(* IEC 61131-3 sources: Std_PalletMover/Class/MQTTClient_Interface (part 5) *)

      pResult^.aData[0]$UDINT := DiagnosticData.ComDiagnosis.udDMEntries;

    //-------------------------------------------------------------
    //TX Rate
    //-------------------------------------------------------------
    MQTTCLIENTINTERFACE_DIAGNOSTIC_NEWINST_GET_TX_RATE:

      pResult^.aData[0]$UDINT := DiagnosticData.ComDiagnosis.udTxRate;

    //-------------------------------------------------------------
    //RX Rate
    //-------------------------------------------------------------
    MQTTCLIENTINTERFACE_DIAGNOSTIC_NEWINST_GET_RX_RATE:

      pResult^.aData[0]$UDINT := DiagnosticData.ComDiagnosis.udRxRate;

    //-------------------------------------------------------------
    //Total RX Bytes
    //-------------------------------------------------------------
    MQTTCLIENTINTERFACE_DIAGNOSTIC_NEWINST_GET_RX_BYTES:

      pResult^.aData[0]$UDINT := DiagnosticData.ComDiagnosis.udTotalBytesRx;

    //-------------------------------------------------------------
    //Total TX Bytes
    //-------------------------------------------------------------
    MQTTCLIENTINTERFACE_DIAGNOSTIC_NEWINST_GET_TX_BYTES:

      pResult^.aData[0]$UDINT := DiagnosticData.ComDiagnosis.udTotalBytesTx;

  end_case;

END_FUNCTION

FUNCTION MQTTClient_Interface::Diagnostic_Event
	VAR_INPUT
		Event 	: t_e_DiagnosticLogTypes;
		udValue 	: UDINT;
	END_VAR

  //==============================================================
  //Based on the event that occurred, change the diagnostic data
  //==============================================================
  case Event of
    //----------------------------------------------------------
    //Reset the Diagnostic Values
    //----------------------------------------------------------
    DL_Reset:

      //Reset the timestamp
      DiagnosticData.udLastCalcTimestamp := ops.tAbsolute;

      //Clear Values
      SigCLib.MemSet( dst :=  #DiagnosticData.ComDiagnosis,
                      c   :=  0x00,
                      len :=  sizeof(DiagnosticData.ComDiagnosis));

      SigCLib.MemSet( dst :=  #DiagnosticData.TransferRateCalc,
                      c   :=  0x00,
                      len :=  sizeof(DiagnosticData.TransferRateCalc));

    //----------------------------------------------------------
    //Increment Connection Count
    //----------------------------------------------------------
    DL_Connect:

      DiagnosticData.ComDiagnosis.udConnect += 1;

    //----------------------------------------------------------
    //Connection Failed
    //----------------------------------------------------------
    DL_ConnectFail:

      DiagnosticData.ComDiagnosis.udConnectFail += 1;

    //----------------------------------------------------------
    //Connection Retried
    //----------------------------------------------------------
    DL_ConnectRetry:

      DiagnosticData.ComDiagnosis.udConnectRetry += 1;

    //----------------------------------------------------------
    //Connection Watchdog Timed out
    //----------------------------------------------------------
    DL_WatchdogTimeout:

      DiagnosticData.ComDiagnosis.udWDTimeout += 1;

    //----------------------------------------------------------
    //NotUsed
    //----------------------------------------------------------
    DL_NotUsed:

    //----------------------------------------------------------
    //Last Error Code Returned from MQTTClient
    //----------------------------------------------------------
    DL_LastErrorCode:

      DiagnosticData.ComDiagnosis.udLastRet := udValue;

    //----------------------------------------------------------
    //Number of errors returned from MQTTClient
    //----------------------------------------------------------
    DL_Error:

      DiagnosticData.ComDiagnosis.udFailRet += 1;

    //----------------------------------------------------------
    //Number of subscribe requests
    //----------------------------------------------------------
    DL_SubRequest:

      DiagnosticData.ComDiagnosis.udSubReqs += 1;

    //----------------------------------------------------------
    //Number of failed subscribe requests
    //----------------------------------------------------------
    DL_SubFail:

      DiagnosticData.ComDiagnosis.udSubFail += 1;

    //----------------------------------------------------------
    //Number of Publish Requests
    //----------------------------------------------------------
    DL_PubRequest:

      DiagnosticData.ComDiagnosis.udPubReq += 1;

    //----------------------------------------------------------
    //Number of failed Publishes
    //----------------------------------------------------------
    DL_PubFail:

      DiagnosticData.ComDiagnosis.udPubFail += 1;

    //----------------------------------------------------------
    //Number of Unsubscribe requests
    //----------------------------------------------------------
    DL_UnsubRequest:

      DiagnosticData.ComDiagnosis.udUnsubReq += 1;

    //----------------------------------------------------------
    //Unsubscribe Failed
    //----------------------------------------------------------
    DL_UnsubFail:

      DiagnosticData.ComDiagnosis.udUnsubFail += 1;

    //----------------------------------------------------------
    //Set PubSubEntries
    //----------------------------------------------------------
    DL_PubSubEntries:

      DiagnosticData.ComDiagnosis.udPubSubEntries := udValue;

    //----------------------------------------------------------
    //Add Log
    //----------------------------------------------------------
    DL_Log:

      DiagnosticData.ComDiagnosis.udLogs += 1;

    //----------------------------------------------------------
    //Ping Request Sent
    //----------------------------------------------------------
    DL_PingReq:

      DiagnosticData.ComDiagnosis.udPingReq += 1;

    //----------------------------------------------------------
    //Ping Response Received
    //----------------------------------------------------------
    DL_PingResp:

      DiagnosticData.ComDiagnosis.udPingResp += 1;

    //----------------------------------------------------------
    //QOS 0 Publish made
    //----------------------------------------------------------
    DL_Pub0:

      DiagnosticData.ComDiagnosis.udPubQOS0 += 1;

    //----------------------------------------------------------
    //QOS1 Publish Made
    //----------------------------------------------------------
    DL_Pub1:

      DiagnosticData.ComDiagnosis.udPubQOS1 += 1;

    //----------------------------------------------------------
    //QOS2 Publish Made
    //----------------------------------------------------------
    DL_Pub2:

      DiagnosticData.ComDiagnosis.udPubQOS2 += 1;

    //----------------------------------------------------------
    //QOS0 Subscribe Made
    //----------------------------------------------------------
    DL_Sub0:

      DiagnosticData.ComDiagnosis.udSubQOS0 += 1;

    //----------------------------------------------------------
    //QOS1 Subscribe Made
    //----------------------------------------------------------
    DL_Sub1:

      DiagnosticData.ComDiagnosis.udSubQOS1 += 1;

    //----------------------------------------------------------
    //QOS2 Subscribe Made
    //----------------------------------------------------------
    DL_Sub2:

      DiagnosticData.ComDiagnosis.udSubQOS2 += 1;

    //----------------------------------------------------------
    //Set DataMap Entries
    //----------------------------------------------------------
    DL_DataMapEntries:

      DiagnosticData.ComDiagnosis.udDMEntries := udValue;

    //----------------------------------------------------------
    //Set TX Rate
    //----------------------------------------------------------
    DL_TXRate:

      DiagnosticData.ComDiagnosis.udTxRate := udValue;

    //----------------------------------------------------------
    //Set RX Rate
    //----------------------------------------------------------
    DL_RXRate:

      DiagnosticData.ComDiagnosis.udRxRate := udValue;

    //----------------------------------------------------------
    //Set RX Bytes
    //----------------------------------------------------------
    DL_RXBytes:

      DiagnosticData.ComDiagnosis.udTotalBytesRx += udValue;

    //----------------------------------------------------------
    //Set TX Bytes
    //----------------------------------------------------------
    DL_TXBytes:

      DiagnosticData.ComDiagnosis.udTotalBytesTx += udValue;

  end_case;

END_FUNCTION

FUNCTION MQTTClient_Interface::ConfigObject_Process
	VAR_OUTPUT
		eRet 	: t_e_TaskRet;
	END_VAR
  VAR
  	ClientIDConfig          : MQTTClient_Interface_ConfigBase::t_s_ClientID;
    ConnectionDetailsConfig : MQTTClient_Interface_ConfigBase::t_s_ConnectionParameters;
    MIMConfig               : MQTTClient_Interface_ConfigBase::t_s_MaxInflightMessages;
    AuthenticationConfig    : MQTTClient_Interface_ConfigBase::t_s_Authentication;
    WillConfig              : MQTTClient_Interface_ConfigBase::t_s_Will;
    ReconnectionConfig      : MQTTClient_Interface_ConfigBase::t_s_ReconnectionParameters;
    TLSConfig               : MQTTClient_Interface_ConfigBase::t_s_TLS;
    tmpPara1                : DINT;
  END_VAR

  //Assume Busy
  eRet := TR_Busy;

  //======================================
  //Proccess the Config Object
  //======================================
  case Config.ConfigObject.State of
    //----------------------------
    //Client ID
    //----------------------------
    CO_ClientID:

      //Call the Config Method
      ClientIDConfig := Config.ConfigObject.pThis$^MQTTClient_Interface_ConfigBase^.ClientID();

      //Check if the config has been made, set the values
      if ClientIDConfig.ClientID <> ACCESS_DENIED then

        //If the input is OK, set the parameters
        if ClientIDConfig.ClientID                                                             &
           SigCLib.StrLen16(str0:=ClientIDConfig.ClientID) < MQTT_PROT_MAX_CLIENTID_NAME_LEN   then

          SigCLib.MemSet( dst   :=  #MQTTClientConfigData.Config.aClientID[0],
                          c     :=  0x00,
                          len   :=  sizeof(MQTTClientConfigData.Config.aClientID));
          SigCLib.StrCpy16(dst0 :=  #MQTTClientConfigData.Config.aClientID[0],
                           src0 :=  ClientIDConfig.ClientID);

          MQTTClientConfigData.Config.bClientIDSet := TRUE;

        //Input Not OK, Log
        else

          Logging_InterfLog(usLevel   :=  MQTTCLIENTINTERFACE_LOGGING_LEVEL_ERR,
                            dMsgGroup :=  MQCLIINF_LOG_ERROR_CONFIG_OBJ_CLIENTID_STRING_LEN_GRP,
                            dMsgNbr   :=  MQCLIINF_LOG_ERROR_CONFIG_OBJ_CLIENTID_STRING_LEN_MSG,
                            pMsg      :=  MQCLIINF_LOG_ERROR_CONFIG_OBJ_CLIENTID_STRING_LEN_TEXT,
                            pPara1    :=  NIL,
                            pPara2    :=  NIL,
                            pPara3    :=  NIL,
                            pPara4    :=  NIL);

        end_if;

      end_if;

      Config.ConfigObject.State := CO_ConnectionDetails;

    //----------------------------
    //Connection Details
    //----------------------------
    CO_ConnectionDetails:

      //Call the Config Method
      ConnectionDetailsConfig := Config.ConfigObject.pThis$^MQTTClient_Interface_ConfigBase^.ConnectionParameters();

      //Check if the config has been made
      if ConnectionDetailsConfig.hostname <> ACCESS_DENIED then

        //If the input is OK, set the parameters
        if ConnectionDetailsConfig.hostname                                                        &
           SigCLib.StrLen16(str0:=ConnectionDetailsConfig.hostname) < MQTTCLIENT_HOSTNAME_MAX_LEN  then

          SigCLib.MemSet( dst   :=  #MQTTClientConfigData.Config.Connect.aHostname[0],
                          c     :=  0x00,
                          len   :=  sizeof(MQTTClientConfigData.Config.Connect.aHostname));
          SigCLib.StrCpy16( dst0  :=  #MQTTClientConfigData.Config.Connect.aHostname[0],
                            src0  :=  ConnectionDetailsConfig.hostname);

          MQTTClientConfigData.Config.Connect.ValuesSet.Hostname := TRUE;

        //Input Not OK, Log
        else

          Logging_InterfLog(usLevel   :=  MQTTCLIENTINTERFACE_LOGGING_LEVEL_ERR,
                            dMsgGroup :=  MQCLIINF_LOG_ERROR_CONFIG_OBJ_HOSTNAME_STR_LEN_GRP,
                            dMsgNbr   :=  MQCLIINF_LOG_ERROR_CONFIG_OBJ_HOSTNAME_STR_LEN_MSG,
                            pMsg      :=  MQCLIINF_LOG_ERROR_CONFIG_OBJ_HOSTNAME_STR_LEN_TEXT,
                            pPara1    :=  NIL,
                            pPara2    :=  NIL,
                            pPara3    :=  NIL,
                            pPara4    :=  NIL);

        end_if;

        //If the input is OK, set the parameters
        if ConnectionDetailsConfig.port > 0       &
           ConnectionDetailsConfig.port <= 65536  then

          MQTTClientConfigData.Config.Connect.iPort := ConnectionDetailsConfig.port;
          MQTTClientConfigData.Config.Connect.ValuesSet.Port := TRUE;

        //Input Not OK, Log
        else

          tmpPara1 := to_dint(ConnectionDetailsConfig.port);

          Logging_InterfLog(usLevel   :=  MQTTCLIENTINTERFACE_LOGGING_LEVEL_ERR,
                            dMsgGroup :=  MQCLIINF_LOG_ERROR_CONFIG_OBJ_PORT_INVALID_GRP,
                            dMsgNbr   :=  MQCLIINF_LOG_ERROR_CONFIG_OBJ_PORT_INVALID_MSG,
                            pMsg      :=  MQCLIINF_LOG_ERROR_CONFIG_OBJ_PORT_INVALID_TEXT,
                            pPara1    :=  #tmpPara1,
                            pPara2    :=  NIL,
                            pPara3    :=  NIL,
                            pPara4    :=  NIL);

        end_if;

        //If the input is OK, set the parameters
        if ConnectionDetailsConfig.keepalive > 0       &
           ConnectionDetailsConfig.keepalive <= 65536  then

          MQTTClientConfigData.Config.Connect.iKeepalive := ConnectionDetailsConfig.keepalive;
          MQTTClientConfigData.Config.Connect.ValuesSet.Keepalive := TRUE;

        //Input Not OK, Log
        else

          tmpPara1 := to_dint(ConnectionDetailsConfig.keepalive);

          Logging_InterfLog(usLevel   :=  MQTTCLIENTINTERFACE_LOGGING_LEVEL_ERR,
                            dMsgGroup :=  MQCLIINF_LOG_ERROR_CONFIG_OBJ_KEEPALIVE_INVALID_GRP,
                            dMsgNbr   :=  MQCLIINF_LOG_ERROR_CONFIG_OBJ_KEEPALIVE_INVALID_MSG,
                            pMsg      :=  MQCLIINF_LOG_ERROR_CONFIG_OBJ_KEEPALIVE_INVALID_TEXT,
                            pPara1    :=  #tmpPara1,
                            pPara2    :=  NIL,
                            pPara3    :=  NIL,
                            pPara4    :=  NIL);

        end_if;

      end_if;

      Config.ConfigObject.State := CO_MaxInflightMessages;

    //----------------------------
    //Max Inflight Messages
    //----------------------------
    CO_MaxInflightMessages:

      //Call the Config Method
      MIMConfig := Config.ConfigObject.pThis$^MQTTClient_Interface_ConfigBase^.MaxInflightMessages();

      //Check if the config has been made
      if MIMConfig.max_inflight_messages <> -1 then

        //If the input is OK, set the parameters
        if MIMConfig.max_inflight_messages >= MQTTCLIENT_MIN_INFLIGHT_MSGS then

          MQTTClientConfigData.Config.Connect.iMaxInflightMessages  := MIMConfig.max_inflight_messages;
          MQTTClientConfigData.Config.Connect.ValuesSet.MaxInflight := TRUE;

        //Input Not OK, Log
        else

          tmpPara1 := MQTTCLIENT_MIN_INFLIGHT_MSGS;

          Logging_InterfLog(usLevel   :=  MQTTCLIENTINTERFACE_LOGGING_LEVEL_ERR,
                            dMsgGroup :=  MQCLIINF_LOG_ERROR_CONFIG_OBJ_MAX_INF_MSGS_LOW_GRP,
                            dMsgNbr   :=  MQCLIINF_LOG_ERROR_CONFIG_OBJ_MAX_INF_MSGS_LOW_MSG,
                            pMsg      :=  MQCLIINF_LOG_ERROR_CONFIG_OBJ_MAX_INF_MSGS_LOW_TEXT,
                            pPara1    :=  #tmpPara1,
                            pPara2    :=  NIL,
                            pPara3    :=  NIL,
                            pPara4    :=  NIL);

        end_if;

      end_if;

      Config.ConfigObject.State := CO_Authentication;

    //----------------------------
    //Authentication
    //----------------------------
    CO_Authentication:

      //Call the Config Method
      AuthenticationConfig := Config.ConfigObject.pThis$^MQTTClient_Interface_ConfigBase^.AuthenticationParameters();

      //Check if the config has been made
      if AuthenticationConfig.username <> ACCESS_DENIED then

        //If the input is OK, set the parameters
        if AuthenticationConfig.username                                                                         &
           SigCLib.StrLen16(str0:=AuthenticationConfig.username) < MQTTCLIENTINTERFACE_CONNECT_USERNAME_MAX_LEN  then

          SigCLib.MemSet( dst   :=  #MQTTClientConfigData.Config.Connect.aUsername[0],
                          c     :=  0x00,
                          len   :=  sizeof(MQTTClientConfigData.Config.Connect.aUsername));
          SigCLib.StrCpy16( dst0  :=  #MQTTClientConfigData.Config.Connect.aUsername[0],
                            src0  :=  AuthenticationConfig.username);

          MQTTClientConfigData.Config.Connect.ValuesSet.Username := TRUE;

        //Input Not OK, Log
        else

          tmpPara1 := MQTTCLIENTINTERFACE_CONNECT_USERNAME_MAX_LEN;

          Logging_InterfLog(usLevel   :=  MQTTCLIENTINTERFACE_LOGGING_LEVEL_ERR,
                            dMsgGroup :=  MQCLIINF_LOG_ERROR_CONFIG_OBJ_AUTH_USN_STR_LEN_GRP,
                            dMsgNbr   :=  MQCLIINF_LOG_ERROR_CONFIG_OBJ_AUTH_USN_STR_LEN_MSG,
                            pMsg      :=  MQCLIINF_LOG_ERROR_CONFIG_OBJ_AUTH_USN_STR_LEN_TEXT,
                            pPara1    :=  #tmpPara1,
                            pPara2    :=  NIL,
                            pPara3    :=  NIL,
                            pPara4    :=  NIL);

          MQTTClientConfigData.Config.Connect.ValuesSet.Username := FALSE;

        end_if;

        //If the input is OK, set the parameters
        if AuthenticationConfig.password                                                                         &
           SigCLib.StrLen16(str0:=AuthenticationConfig.password) < MQTTCLIENTINTERFACE_CONNECT_PASSWORD_MAX_LEN  then

          SigCLib.MemSet( dst   :=  #MQTTClientConfigData.Config.Connect.aPassword[0],
                          c     :=  0x00,
                          len   :=  sizeof(MQTTClientConfigData.Config.Connect.aPassword));
          SigCLib.StrCpy16( dst0  :=  #MQTTClientConfigData.Config.Connect.aPassword[0],
                            src0  :=  AuthenticationConfig.password);

          MQTTClientConfigData.Config.Connect.ValuesSet.Password := TRUE;

        //Input Not OK, Log
        else

          tmpPara1 := MQTTCLIENTINTERFACE_CONNECT_PASSWORD_MAX_LEN;

          Logging_InterfLog(usLevel   :=  MQTTCLIENTINTERFACE_LOGGING_LEVEL_ERR,
                            dMsgGroup :=  MQCLIINF_LOG_ERROR_CONFIG_OBJ_AUTH_PASS_STR_LEN_GRP,
                            dMsgNbr   :=  MQCLIINF_LOG_ERROR_CONFIG_OBJ_AUTH_PASS_STR_LEN_MSG,
                            pMsg      :=  MQCLIINF_LOG_ERROR_CONFIG_OBJ_AUTH_PASS_STR_LEN_TEXT,
                            pPara1    :=  #tmpPara1,
                            pPara2    :=  NIL,
                            pPara3    :=  NIL,
                            pPara4    :=  NIL);

          MQTTClientConfigData.Config.Connect.ValuesSet.Password := FALSE;

        end_if;

      end_if;

      Config.ConfigObject.State := CO_Will;

    //----------------------------
    //Will Config
    //----------------------------
    CO_Will:

      //Call the Config Method
      WillConfig := Config.ConfigObject.pThis$^MQTTClient_Interface_ConfigBase^.Will();

      //Check if the config has been made
      if WillConfig.topic <> ACCESS_DENIED then

        //If the input is OK, set the parameters
        if WillConfig.topic                                                                   &
           SigCLib.StrLen16(str0:=WillConfig.topic) < MQTTCLIENTINTERFACE_WILL_TOPIC_MAX_LEN  then

          SigCLib.MemSet( dst   :=  #MQTTClientConfigData.Config.Will.aTopic[0],
                          c     :=  0x00,
                          len   :=  sizeof(MQTTClientConfigData.Config.Will.aTopic));
          SigCLib.StrCpy16( dst0  :=  #MQTTClientConfigData.Config.Will.aTopic[0],
                            src0  :=  WillConfig.topic);

          MQTTClientConfigData.Config.Will.ValuesSet.Topic := TRUE;

        //Input Not OK, Log
        else

          tmpPara1 := MQTTCLIENTINTERFACE_WILL_TOPIC_MAX_LEN;

          Logging_InterfLog(usLevel   :=  MQTTCLIENTINTERFACE_LOGGING_LEVEL_ERR,
                            dMsgGroup :=  MQCLIINF_LOG_ERROR_CONFIG_OBJ_WILL_TOPIC_STR_LEN_GRP,
                            dMsgNbr   :=  MQCLIINF_LOG_ERROR_CONFIG_OBJ_WILL_TOPIC_STR_LEN_MSG,
                            pMsg      :=  MQCLIINF_LOG_ERROR_CONFIG_OBJ_WILL_TOPIC_STR_LEN_TEXT,
                            pPara1    :=  #tmpPara1,
                            pPara2    :=  NIL,
                            pPara3    :=  NIL,
                            pPara4    :=  NIL);

        end_if;

        //If the input is OK, set the parameters
        if WillConfig.payloadtext                                                                  &
           SigCLib.StrLen(str:=WillConfig.payloadtext) < MQTTCLIENTINTERFACE_WILL_PAYLOAD_MAX_LEN  then

          SigCLib.MemSet( dst   :=  #MQTTClientConfigData.Config.Will.aPayload[0],
                          c     :=  0x00,
                          len   :=  sizeof(MQTTClientConfigData.Config.Will.aPayload));
          SigCLib.StrCpy( dst0  :=  #MQTTClientConfigData.Config.Will.aPayload[0],
                          src0  :=  WillConfig.payloadtext);

          MQTTClientConfigData.Config.Will.ValuesSet.Payload := TRUE;

        //Input Not OK, Log
        else

          tmpPara1 := MQTTCLIENTINTERFACE_WILL_PAYLOAD_MAX_LEN;

          Logging_InterfLog(usLevel   :=  MQTTCLIENTINTERFACE_LOGGING_LEVEL_ERR,
                            dMsgGroup :=  MQCLIINF_LOG_ERROR_CONFIG_OBJ_WILL_PAYLOAD_STR_LEN_GRP,
                            dMsgNbr   :=  MQCLIINF_LOG_ERROR_CONFIG_OBJ_WILL_PAYLOAD_STR_LEN_MSG,
                            pMsg      :=  MQCLIINF_LOG_ERROR_CONFIG_OBJ_WILL_PAYLOAD_STR_LEN_TEXT,
                            pPara1    :=  #tmpPara1,
                            pPara2    :=  NIL,
                            pPara3    :=  NIL,
                            pPara4    :=  NIL);

        end_if;

        //If the input is OK, set the parameters
        if WillConfig.qos >= MQTT_PROT_QOS_MIN  &
           WillConfig.qos <= MQTT_PROT_QOS_MAX  then

          MQTTClientConfigData.Config.Will.iQoS := WillConfig.qos;
          MQTTClientConfigData.Config.Will.ValuesSet.QoS := TRUE;

        //Input Not OK, Log
        else

          tmpPara1 := to_dint(WillConfig.qos);

          Logging_InterfLog(usLevel   :=  MQTTCLIENTINTERFACE_LOGGING_LEVEL_ERR,
                            dMsgGroup :=  MQCLIINF_LOG_ERROR_CONFIG_OBJ_WILL_QOS_INVALID_GRP,
                            dMsgNbr   :=  MQCLIINF_LOG_ERROR_CONFIG_OBJ_WILL_QOS_INVALID_MSG,
                            pMsg      :=  MQCLIINF_LOG_ERROR_CONFIG_OBJ_WILL_QOS_INVALID_TEXT,
                            pPara1    :=  #tmpPara1,
                            pPara2    :=  NIL,
                            pPara3    :=  NIL,
                            pPara4    :=  NIL);

        end_if;

        //Retain has an exclusive state choice.
        MQTTClientConfigData.Config.Will.bRetain := WillConfig.bRetain;
        MQTTClientConfigData.Config.Will.ValuesSet.RetainWill := TRUE;

      end_if;

      Config.ConfigObject.State := CO_Reconnection;

    //----------------------------
    //Reconnection Parameters
    //----------------------------
    CO_Reconnection:

      //Call the Config Method
      ReconnectionConfig := Config.ConfigObject.pThis$^MQTTClient_Interface_ConfigBase^.ReconnectionParameters();

      //Check if the config has been made
      if ReconnectionConfig.min_interval <> -1 then

        //If the input is OK, set the parameters
        if ReconnectionConfig.min_interval >= 0                               &
           ReconnectionConfig.min_interval < ReconnectionConfig.max_interval  then

          MQTTClientConfigData.Config.Reconnect.iMinInterval          := ReconnectionConfig.min_interval;
          MQTTClientConfigData.Config.Reconnect.ValuesSet.MinInterval := TRUE;

        //Input Not OK, Log
        else

          Logging_InterfLog(usLevel   :=  MQTTCLIENTINTERFACE_LOGGING_LEVEL_ERR,
                            dMsgGroup :=  MQCLIINF_LOG_ERROR_CONFIG_OBJ_RECONN_MIN_TIME_INVALID_GRP,
                            dMsgNbr   :=  MQCLIINF_LOG_ERROR_CONFIG_OBJ_RECONN_MIN_TIME_INVALID_MSG,
                            pMsg      :=  MQCLIINF_LOG_ERROR_CONFIG_OBJ_RECONN_MIN_TIME_INVALID_TEXT,
                            pPara1    :=  NIL,
                            pPara2    :=  NIL,
                            pPara3    :=  NIL,
                            pPara4    :=  NIL);

        end_if;

        //If the input is OK, set the parameters
        if ReconnectionConfig.max_interval >= 0                               &
           ReconnectionConfig.max_interval > ReconnectionConfig.min_interval  then

          MQTTClientConfigData.Config.Reconnect.iMaxInterval := ReconnectionConfig.max_interval;
          MQTTClientConfigData.Config.Reconnect.ValuesSet.MaxInterval := TRUE;

        //Input Not OK, Log
        else

          Logging_InterfLog(usLevel   :=  MQTTCLIENTINTERFACE_LOGGING_LEVEL_ERR,
                            dMsgGroup :=  MQCLIINF_LOG_ERROR_CONFIG_OBJ_RECONN_MAX_TIME_INVALID_GRP,
                            dMsgNbr   :=  MQCLIINF_LOG_ERROR_CONFIG_OBJ_RECONN_MAX_TIME_INVALID_MSG,
                            pMsg      :=  MQCLIINF_LOG_ERROR_CONFIG_OBJ_RECONN_MAX_TIME_INVALID_TEXT,
                            pPara1    :=  NIL,
                            pPara2    :=  NIL,
                            pPara3    :=  NIL,
                            pPara4    :=  NIL);

        end_if;

        //Scale has an exclusive state choice.
        MQTTClientConfigData.Config.Reconnect.bExponential                := ReconnectionConfig.exponential_scale;
        MQTTClientConfigData.Config.Reconnect.ValuesSet.ExponentialScale  := TRUE;

      end_if;

      Config.ConfigObject.State := CO_TLS;

    //----------------------------
    //TLS Config
    //----------------------------
    CO_TLS:

      //Call the Config Method
      TLSConfig := Config.ConfigObject.pThis$^MQTTClient_Interface_ConfigBase^.TLS();

      //Check if the config has been made
      if TLSConfig.cafile <> ACCESS_DENIED then

        //Se the TLS ValuesSet Flag
        MQTTClientConfigData.Config.TLS.ValuesSet.TLS := TRUE;

        //If the input is OK, set the parameters
        if TLSConfig.cafile then

          if SigCLib.StrLen(str:=TLSConfig.cafile) < MQTTCLIENTINTERFACE_TLS_CAFILE_MAX_LEN  then

            SigCLib.MemSet( dst   :=  #MQTTClientConfigData.Config.TLS.aCAFile[0],
                            c     :=  0x00,
                            len   :=  sizeof(MQTTClientConfigData.Config.TLS.aCAFile));
            SigCLib.StrCpy( dst0   :=  #MQTTClientConfigData.Config.TLS.aCAFile[0],
                            src0   :=  TLSConfig.cafile);

            MQTTClientConfigData.Config.TLS.ValuesSet.CAFile := TRUE;

          //Input Not OK, Log
          else

            tmpPara1 := MQTTCLIENTINTERFACE_TLS_CAFILE_MAX_LEN;

            Logging_InterfLog(usLevel   :=  MQTTCLIENTINTERFACE_LOGGING_LEVEL_ERR,
                              dMsgGroup :=  MQCLIINF_LOG_ERROR_CONFIG_OBJ_TLS_CAFILE_STR_LEN_GRP,
                              dMsgNbr   :=  MQCLIINF_LOG_ERROR_CONFIG_OBJ_TLS_CAFILE_STR_LEN_MSG,
                              pMsg      :=  MQCLIINF_LOG_ERROR_CONFIG_OBJ_TLS_CAFILE_STR_LEN_TEXT,
                              pPara1    :=  #tmpPara1,
                              pPara2    :=  NIL,
                              pPara3    :=  NIL,
                              pPara4    :=  NIL);

          end_if;

        end_if;

        //If the input is OK, set the parameters
        if TLSConfig.certfile then

          if SigCLib.StrLen(str:=TLSConfig.certfile) < MQTTCLIENTINTERFACE_TLS_CERTFILE_MAX_LEN then

            SigCLib.MemSet( dst   :=  #MQTTClientConfigData.Config.TLS.aCertFile[0],
                            c     :=  0x00,
                            len   :=  sizeof(MQTTClientConfigData.Config.TLS.aCertFile));
            SigCLib.StrCpy( dst0   :=  #MQTTClientConfigData.Config.TLS.aCertFile[0],
                            src0   :=  TLSConfig.certfile);

            MQTTClientConfigData.Config.TLS.ValuesSet.CertFile := TRUE;

          //Input Not OK, Log
          else

            tmpPara1 := MQTTCLIENTINTERFACE_TLS_CERTFILE_MAX_LEN;

            Logging_InterfLog(usLevel   :=  MQTTCLIENTINTERFACE_LOGGING_LEVEL_ERR,
                              dMsgGroup :=  MQCLIINF_LOG_ERROR_CONFIG_OBJ_TLS_CERTFILE_STR_LEN_GRP,
                              dMsgNbr   :=  MQCLIINF_LOG_ERROR_CONFIG_OBJ_TLS_CERTFILE_STR_LEN_MSG,
                              pMsg      :=  MQCLIINF_LOG_ERROR_CONFIG_OBJ_TLS_CERTFILE_STR_LEN_TEXT,
                              pPara1    :=  #tmpPara1,
                              pPara2    :=  NIL,
                              pPara3    :=  NIL,
                              pPara4    :=  NIL);

          end_if;

        end_if;

        //If the input is OK, set the parameters
        if TLSConfig.keyfile then

          if SigCLib.StrLen(str:=TLSConfig.keyfile) < MQTTCLIENTINTERFACE_TLS_KEYFILE_MAX_LEN then

            SigCLib.MemSet( dst   :=  #MQTTClientConfigData.Config.TLS.aKeyFile[0],
                            c     :=  0x00,
                            len   :=  sizeof(MQTTClientConfigData.Config.TLS.aKeyFile));
            SigCLib.StrCpy(dst0    :=  #MQTTClientConfigData.Config.TLS.aKeyFile[0],
                           src0    :=  TLSConfig.keyfile);

            MQTTClientConfigData.Config.TLS.ValuesSet.KeyFile := TRUE;

          //Input Not OK, Log
          else

            tmpPara1 := MQTTCLIENTINTERFACE_TLS_KEYFILE_MAX_LEN;

            Logging_InterfLog(usLevel   :=  MQTTCLIENTINTERFACE_LOGGING_LEVEL_ERR,
                              dMsgGroup :=  MQCLIINF_LOG_ERROR_CONFIG_OBJ_TLS_KEYFILE_STR_LEN_GRP,
                              dMsgNbr   :=  MQCLIINF_LOG_ERROR_CONFIG_OBJ_TLS_KEYFILE_STR_LEN_MSG,
                              pMsg      :=  MQCLIINF_LOG_ERROR_CONFIG_OBJ_TLS_KEYFILE_STR_LEN_TEXT,
                              pPara1    :=  #tmpPara1,
                              pPara2    :=  NIL,
                              pPara3    :=  NIL,
                              pPara4    :=  NIL);

          end_if;

        end_if;

        //If the input is OK, set the parameters
        if TLSConfig.pw then

          if SigCLib.StrLen(str:=TLSConfig.pw) < MQTTCLIENTINTERFACE_TLS_PASSWORD_MAX_LEN then

            SigCLib.MemSet( dst   :=  #MQTTClientConfigData.Config.TLS.aPassword[0],
                            c     :=  0x00,
                            len   :=  sizeof(MQTTClientConfigData.Config.TLS.aPassword));
            SigCLib.StrCpy( dst0   :=  #MQTTClientConfigData.Config.TLS.aPassword[0],
                            src0   :=  TLSConfig.pw);

            MQTTClientConfigData.Config.TLS.ValuesSet.Password := TRUE;

          //Input Not OK, Log
          else

            tmpPara1 := MQTTCLIENTINTERFACE_TLS_PASSWORD_MAX_LEN;

            Logging_InterfLog(usLevel   :=  MQTTCLIENTINTERFACE_LOGGING_LEVEL_ERR,
                              dMsgGroup :=  MQCLIINF_LOG_ERROR_CONFIG_OBJ_TLS_PASS_STR_LEN_GRP,
                              dMsgNbr   :=  MQCLIINF_LOG_ERROR_CONFIG_OBJ_TLS_PASS_STR_LEN_MSG,
                              pMsg      :=  MQCLIINF_LOG_ERROR_CONFIG_OBJ_TLS_PASS_STR_LEN_TEXT,
                              pPara1    :=  #tmpPara1,
                              pPara2    :=  NIL,
                              pPara3    :=  NIL,
                              pPara4    :=  NIL);

          end_if;

        end_if;

      end_if;

      Config.ConfigObject.State := CO_ClientID;
      eRet := TR_Done;

  end_case;

END_FUNCTION

FUNCTION GLOBAL MQTTClient_Interface::Config_Login
	VAR_INPUT
		pThis 	: ^void;
	END_VAR
	VAR_OUTPUT
		bOK 	: BOOL;
	END_VAR

  //If the pointer is not OK, stop
  if pThis = NIL then
    bOK := FALSE;
    return;
  end_if;

  //If the Login has been set before, fail, else accept
  if Config.ConfigObject.pThis then
    bOK := FALSE;
  else
    bOK := TRUE;
    Config.ConfigObject.pThis := pThis;
  end_if;

END_FUNCTION

FUNCTION MQTTClient_Interface::Diagnostic_ReadErrors
  VAR
  	udErr : UDINT;
    pErrStr : ^CHAR;
  END_VAR

  //If a sufficient amount of time has passed, check for errors
  if ops.tAbsolute - DiagnosticData.udLastErrorCheck >= MQTTCLIENTINTERFACE_DIAGNOSTIC_ERROR_CHECK_INTERVAL then

    //Update timestamp
    DiagnosticData.udLastErrorCheck := ops.tAbsolute;

    //If SSL is activated, check the interface for errors
    if MQTTClientConfigData.Config.TLS.ValuesSet.TLS then

      udErr := OpenSSL.ERR_get_error();

      if udErr <> 0 then

        pErrStr := OpenSSL.ERR_error_string(e   :=  udErr,
                                            buf :=  NIL);

        if pErrStr then

          Logging_InterfLog(usLevel     :=  MQTT_LOG_ERR,
                            dMsgGroup   :=  MQTTCLIENT_INTERFACE_LOG_ERROR_OPENSSL_MSGGROUP,
                            dMsgNbr     :=  to_dint(udErr),
                            pMsg        :=  pErrStr,
                            pPara1      :=  NIL,
                            pPara2      :=  NIL,
                            pPara3      :=  NIL,
                            pPara4      :=  NIL);

        end_if;

      end_if;

    end_if;

  end_if;

END_FUNCTION

FUNCTION GLOBAL MQTTClient_Interface::Config_SetParameter
	VAR_INPUT
		Parameter 	: t_e_ConfigParameters;
		Value 	: DINT;
	END_VAR
	VAR_OUTPUT
		retCode 	: INT;
	END_VAR

  //Assume OK
  retCode := 0;

  //===============================================================
  //Based on the selected Parameter, attempt to change the setting
  //===============================================================
  case Parameter of

    //-------------------------------------------
    //Sets whether the DataMap publishes OnChange
    //values when added or waits for first change
    //-------------------------------------------
  	t_e_ConfigParameters::CP_DataMap_SendOnAdd:

      //Valid
      if Value = 0 | Value = 1 then

        if Config.pDataMapConfig <> NIL then
          Config.pDataMapConfig^.Config.bSendOnAdd := (Value = 1);
        end_if;

      //Invalid
      else

        retCode := MQTTClient::MQTT_ERR_INVAL;

      end_if;

  end_case;

END_FUNCTION
